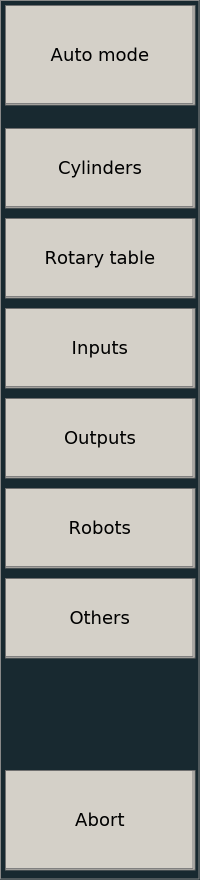
VISUALIZATION NavBarManual  // 200x880
VAR_IN_OUT
	btnAutoMode	: BOOL;
	btnCylinders: BOOL;
	btnMotors	: BOOL;
	btnSafety	: BOOL;
	btnInputs	: BOOL;
	btnOutputs	: BOOL;
	btnOthers	: BOOL;
	btnAbort	: BOOL;
	btnRobots 	: BOOL;
END_VAR
    Button (5,128 190x80), "Cylinders", invisible if: TRUE, input disabled if: TRUE
        tap btnCylinders
    Button (5,218 190x80), "Rotary table"
        tap btnMotors
    Button (5,770 190x100), "Abort"
        tap btnAbort
    Button (5,398 190x80), "Outputs"
        tap btnOutputs
    Button (5,308 190x80), "Inputs"
        tap btnInputs
    Button (5,5 190x100), "Auto mode"
        tap btnAutoMode
    Button (5,578 190x80), "Others"
        tap btnOthers
    Button (5,488 190x80), "Robots"
        tap btnRobots
END_VISUALIZATION

(* stored: Version 1.1.0.1, ProductVersion 3.1.4024.9
   Visu NavBarManual: Id {da2fcb43-3c28-4c3b-ab2b-9fca12895bcd} *)
